// TIA Portal V16 export
// export: Created 2021-04-06T19:52:15.2153199Z, ExportSetting WithDefaults, DisplayName Totally Integrated Automation Portal, DisplayVersion V16, DisplayName TIA Portal Version Control Interface, DisplayVersion V16, DisplayName TIA Portal Openness, DisplayVersion V16, DisplayName STEP 7 Professional, DisplayVersion V16, DisplayName STEP 7 Safety, DisplayVersion V16, DisplayName WinCC Unified SCADA Engineering System, DisplayVersion V16
FUNCTION_BLOCK "modbus_SenecaConnectPort1"   // FB11, LAD
{ S7_Optimized_Access := 'TRUE' }
VERSION : 0.1
// stored: AutoNumber true, IsIECCheckEnabled false, IsRetainMemResEnabled false, MemoryReserve 100, SetENOAutomatically false, UDAEnableTagReadback false
   VAR_INPUT
      port : PORT;   // порт для подключения
      arrayAddressModbus : Array[0..12] of UInt;
      Offset_array_bits : SInt;
   END_VAR
   VAR_IN_OUT
      calibrateZero : Array[0..12] of Bool;
      taraZero : Array[0..12] of Bool;
      currentWeight : Array[0..12] of Real;
   END_VAR
   VAR
      MB_COMM_LOAD { S7_SetPoint := 'True'} : MB_COMM_LOAD;
      MB_MASTER { S7_SetPoint := 'True'} : MB_MASTER;
      Seneca : Struct
         TON_changeStep : TON_TIME;
         TON_Start { S7_SetPoint := 'True'} : Bool;
         "Step" : SInt;
      END_STRUCT;
      tmpWeight : Array[0..12] of DWord;
      restartPort : Bool;   // перезагрузка Modbus
   END_VAR
   VAR_TEMP
      index : SInt;
      tmpIndex : SInt;
   END_VAR
BEGIN

REGION Network 1: ИНИЦИАЛИЗИРУЕМ ПОРТ
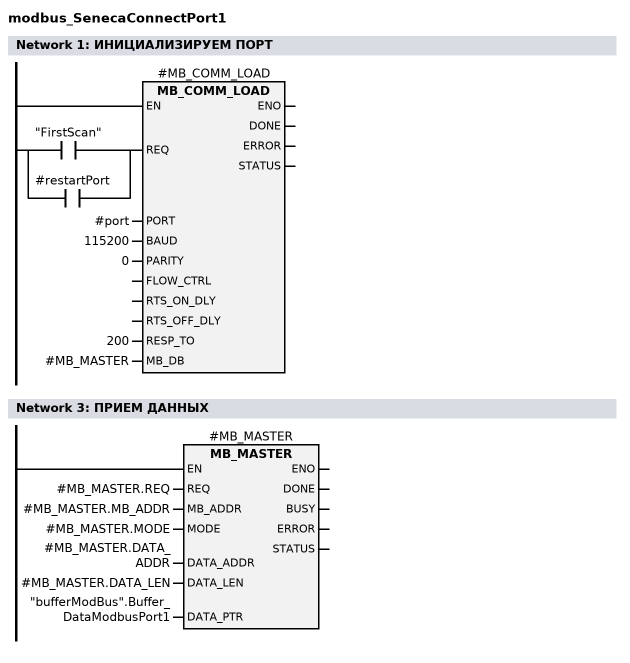
   RUNG wire#powerrail
      #MB_COMM_LOAD.MB_COMM_LOAD(REQ := wire#w1, PORT := #port, BAUD := 115200, PARITY := 0, FLOW_CTRL :=, RTS_ON_DLY :=, RTS_OFF_DLY :=, RESP_TO := 200, MB_DB := #MB_MASTER, DONE =>, ERROR =>, STATUS =>)
   END_RUNG
   RUNG wire#powerrail
      Contact( "FirstScan" )
   END_RUNG wire#w1
   RUNG wire#powerrail
      Contact( #restartPort )
   END_RUNG wire#w1
   // the same network as SCL:
   #MB_COMM_LOAD(REQ := "FirstScan" OR #restartPort,   // MB_COMM_LOAD
                 PORT := #port,
                 BAUD := 115200,
                 PARITY := 0,
                 RESP_TO := 200,
                 MB_DB := #MB_MASTER);
END_REGION

REGION Network 2 (SCL): ОБМЕН
   #Seneca.TON_changeStep(IN :=#Seneca.TON_Start,
                          PT := t#15ms);

   CASE #Seneca.Step OF

       1:
           #Seneca.Step := #Seneca.Step + 1;

       2: //ЧИТАЕМ ЗНАЧЕНИЕ ВЕСА С ПЕРВОГО МОДУЛЯ

           #index := 1+#Offset_array_bits;//заполнять функцию будем через индекс чтобы меньше писать
           "rcvDataWeight"(ADDR_DEVICE := #arrayAddressModbus[#index],
                           Ton_changeStep:=#Seneca.TON_changeStep,
                           Ton_Start:=#Seneca.TON_Start,
                           "Step":=#Seneca.Step,
                           MB_MASTER:=#MB_MASTER);

       3://ЧИТАЕМ ЗНАЧЕНИЕ ВЕСА СО ВТОРОГО МОДУЛЯ
           #index := 2+#Offset_array_bits;//заполнять функцию будем через индекс чтобы меньше писать
           "rcvDataWeight"(ADDR_DEVICE := #arrayAddressModbus[#index],
                           Ton_changeStep:=#Seneca.TON_changeStep,
                           Ton_Start:=#Seneca.TON_Start,
                           "Step":=#Seneca.Step,
                           MB_MASTER:=#MB_MASTER);

       4: // КАЛИБРОВКА 0 ДЛЯ ПЕРВОГО МОДУЛЯ и ТАРИРОВАНИЕ
           #index := 1+#Offset_array_bits;//заполнять функцию будем через индекс чтобы меньше писать
           "sndCALIBR&Tara"(ADDR_DEVICE := #arrayAddressModbus[#index],
                        ton_changeStep:=#Seneca.TON_changeStep,
                        MB_MASTER:=#MB_MASTER,
                        Ton_Start:=#Seneca.TON_Start,
                        Calibrate:=#calibrateZero[#index],
                        Buffer:="bufferModBus".Buffer_DataModbusPort1,
                        "Step":=#Seneca.Step,
                        Tara:=#taraZero[#index]);

       5:// КАЛИБРОВКА 0 ДЛЯ ВТОРОГО МОДУЛЯ и ТАРИРОВАНИЕ
           #index := 2+#Offset_array_bits;//заполнять функцию будем через индекс чтобы меньше писать
           "sndCALIBR&Tara"(ADDR_DEVICE := #arrayAddressModbus[#index],
                        ton_changeStep := #Seneca.TON_changeStep,
                        MB_MASTER := #MB_MASTER,
                        Ton_Start := #Seneca.TON_Start,
                        Calibrate := #calibrateZero[#index],
                        Buffer := "bufferModBus".Buffer_DataModbusPort1,
                        "Step" := #Seneca.Step,
                        Tara := #taraZero[#index]);

           //////////////////////////////////////////////////////////////////////////////////
           //////////////////////////////////////////////////////////////////////////////////
           //////////////////////////////////////////////////////////////////////////////////
           //////////////////////////////////////////////////////////////////////////////////
       6: //ЧИТАЕМ ЗНАЧЕНИЕ ВЕСА С ТРЕТЬЕГО МОДУЛЯ

           #index := 3+#Offset_array_bits;//заполнять функцию будем через индекс чтобы меньше писать
           "rcvDataWeight"(ADDR_DEVICE := #arrayAddressModbus[#index],
                           Ton_changeStep := #Seneca.TON_changeStep,
                           Ton_Start := #Seneca.TON_Start,
                           "Step" := #Seneca.Step,
                           MB_MASTER := #MB_MASTER);

       7://ЧИТАЕМ ЗНАЧЕНИЕ ВЕСА С ЧЕТВЕРТОГО МОДУЛЯ
           #index := 4+#Offset_array_bits;//заполнять функцию будем через индекс чтобы меньше писать
           "rcvDataWeight"(ADDR_DEVICE := #arrayAddressModbus[#index],
                           Ton_changeStep := #Seneca.TON_changeStep,
                           Ton_Start := #Seneca.TON_Start,
                           "Step" := #Seneca.Step,
                           MB_MASTER := #MB_MASTER);

       8:// КАЛИБРОВКА 0 ДЛЯ ТРЕТЬЕГО  МОДУЛЯ

           #index := 3+#Offset_array_bits;//заполнять функцию будем через индекс чтобы меньше писать
           "sndCALIBR&Tara"(ADDR_DEVICE := #arrayAddressModbus[#index],
                        ton_changeStep := #Seneca.TON_changeStep,
                        MB_MASTER := #MB_MASTER,
                        Ton_Start := #Seneca.TON_Start,
                        Calibrate := #calibrateZero[#index],
                        Buffer := "bufferModBus".Buffer_DataModbusPort1,
                        "Step" := #Seneca.Step,
                        Tara := #taraZero[#index]);

       9://КАЛИБРОВКА 0 ДЛЯ ЧЕТВЕРТОГО МОДУЛЯ

           #index := 4+#Offset_array_bits;//заполнять функцию будем через индекс чтобы меньше писать
           "sndCALIBR&Tara"(ADDR_DEVICE := #arrayAddressModbus[#index],
                        ton_changeStep := #Seneca.TON_changeStep,
                        MB_MASTER := #MB_MASTER,
                        Ton_Start := #Seneca.TON_Start,
                        Calibrate := #calibrateZero[#index],
                        Buffer := "bufferModBus".Buffer_DataModbusPort1,
                        "Step" := #Seneca.Step,
                        Tara := #taraZero[#index]);

           /////////////////////////////////////////////////////////////////////////////////
           ////////////////////////////////////////////////////////////////////////////////
           ////////////////////////////////////////////////////////////////////////////////
           ////////////////////////////////////////////////////////////////////////////////
       10: //ЧИТАЕМ ЗНАЧЕНИЕ ВЕСА С ПЯТОГО МОДУЛЯ
           #index := 5+#Offset_array_bits;//заполнять функцию будем через индекс чтобы меньше писать
           "rcvDataWeight"(ADDR_DEVICE := #arrayAddressModbus[#index],
                           Ton_changeStep := #Seneca.TON_changeStep,
                           Ton_Start := #Seneca.TON_Start,
                           "Step" := #Seneca.Step,
                           MB_MASTER := #MB_MASTER);

       11://ЧИТАЕМ ЗНАЧЕНИЕ ВЕСА С ШЕСТОГО МОДУЛЯ
           #index := 6+#Offset_array_bits;//заполнять функцию будем через индекс чтобы меньше писать
           "rcvDataWeight"(ADDR_DEVICE := #arrayAddressModbus[#index],
                           Ton_changeStep := #Seneca.TON_changeStep,
                           Ton_Start := #Seneca.TON_Start,
                           "Step" := #Seneca.Step,
                           MB_MASTER := #MB_MASTER);

       12:// КАЛИБРОВКА 0 ДЛЯ ПЯТОГО  МОДУЛЯ

           #index := 5+#Offset_array_bits;//заполнять функцию будем через индекс чтобы меньше писать
           "sndCALIBR&Tara"(ADDR_DEVICE := #arrayAddressModbus[#index],
                        ton_changeStep := #Seneca.TON_changeStep,
                        MB_MASTER := #MB_MASTER,
                        Ton_Start := #Seneca.TON_Start,
                        Calibrate := #calibrateZero[#index],
                        Buffer := "bufferModBus".Buffer_DataModbusPort1,
                        "Step" := #Seneca.Step,
                        Tara := #taraZero[#index]);

       13:// КАЛИБРОВКА 0 ДЛЯ ШЕСТОГО МОДУЛЯ
           #index := 6+#Offset_array_bits;//заполнять функцию будем через индекс чтобы меньше писать
           "sndCALIBR&Tara"(ADDR_DEVICE := #arrayAddressModbus[#index],
                        ton_changeStep := #Seneca.TON_changeStep,
                        MB_MASTER := #MB_MASTER,
                        Ton_Start := #Seneca.TON_Start,
                        Calibrate := #calibrateZero[#index],
                        Buffer := "bufferModBus".Buffer_DataModbusPort1,
                        "Step" := #Seneca.Step,
                        Tara := #taraZero[#index]);
   14://отправка аналоговых значений вибрации
       "sndVibration"(ADDR_DEVICE:=40,
                      ton_changeStep:= #Seneca.TON_changeStep,
                      MB_MASTER:=#MB_MASTER,
                      Ton_Start:=#Seneca.TON_Start,
                      Buffer:="bufferModBus".Buffer_DataModbusPort1,
                      "Step":=#Seneca.Step);

       ELSE
           #Seneca.Step := 1;
   END_CASE;
END_REGION

REGION Network 3: ПРИЕМ ДАННЫХ
   RUNG wire#powerrail
      #MB_MASTER.MB_MASTER(REQ := #MB_MASTER.REQ, MB_ADDR := #MB_MASTER.MB_ADDR, MODE := #MB_MASTER.MODE, DATA_ADDR := #MB_MASTER.DATA_ADDR, DATA_LEN := #MB_MASTER.DATA_LEN, DATA_PTR := "bufferModBus".Buffer_DataModbusPort1, DONE =>, BUSY =>, ERROR =>, STATUS =>)
   END_RUNG
   // the same network as SCL:
   #MB_MASTER(REQ := #MB_MASTER.REQ,   // MB_MASTER
              MB_ADDR := #MB_MASTER.MB_ADDR,
              MODE := #MB_MASTER.MODE,
              DATA_ADDR := #MB_MASTER.DATA_ADDR,
              DATA_LEN := #MB_MASTER.DATA_LEN,
              DATA_PTR := "bufferModBus".Buffer_DataModbusPort1);
END_REGION

REGION Network 4 (SCL)
   IF #Seneca.Step = 2 AND #MB_MASTER.DONE THEN
       #tmpIndex := 1 + #Offset_array_bits;
       #tmpWeight[#tmpIndex].%W0 := "bufferModBus".Buffer_DataModbusPort1[1];
       #tmpWeight[#tmpIndex].%W1 := "bufferModBus".Buffer_DataModbusPort1[0];
       #currentWeight[#tmpIndex] := DWORD_TO_REAL(#tmpWeight[#tmpIndex]);
       "bufferModBus".Buffer_DataModbusPort1[0] := 0;
       "bufferModBus".Buffer_DataModbusPort1[1] := 0;

   END_IF;

   IF #Seneca.Step = 3 AND #MB_MASTER.DONE THEN
       #tmpIndex := 2 + #Offset_array_bits;
       #tmpWeight[#tmpIndex].%W0 := "bufferModBus".Buffer_DataModbusPort1[1];
       #tmpWeight[#tmpIndex].%W1 := "bufferModBus".Buffer_DataModbusPort1[0];
       #currentWeight[#tmpIndex] := DWORD_TO_REAL(#tmpWeight[#tmpIndex]);
       "bufferModBus".Buffer_DataModbusPort1[0] := 0;
       "bufferModBus".Buffer_DataModbusPort1[1] := 0;
   END_IF;

   IF #Seneca.Step = 6 AND #MB_MASTER.DONE THEN
       #tmpIndex := 3 + #Offset_array_bits;
       #tmpWeight[#tmpIndex].%W0 := "bufferModBus".Buffer_DataModbusPort1[1];
       #tmpWeight[#tmpIndex].%W1 := "bufferModBus".Buffer_DataModbusPort1[0];
       #currentWeight[#tmpIndex] := DWORD_TO_REAL(#tmpWeight[#tmpIndex]);
       "bufferModBus".Buffer_DataModbusPort1[0] := 0;
       "bufferModBus".Buffer_DataModbusPort1[1] := 0;
   END_IF;

   IF #Seneca.Step = 7 AND #MB_MASTER.DONE THEN
       #tmpIndex := 4 + #Offset_array_bits;
       #tmpWeight[#tmpIndex].%W0 := "bufferModBus".Buffer_DataModbusPort1[1];
       #tmpWeight[#tmpIndex].%W1 := "bufferModBus".Buffer_DataModbusPort1[0];
       #currentWeight[#tmpIndex] := DWORD_TO_REAL(#tmpWeight[#tmpIndex]);
       "bufferModBus".Buffer_DataModbusPort1[0] := 0;
       "bufferModBus".Buffer_DataModbusPort1[1] := 0;
   END_IF;

   IF #Seneca.Step = 10 AND #MB_MASTER.DONE THEN
       #tmpIndex := 5 + #Offset_array_bits;
       #tmpWeight[#tmpIndex].%W0 := "bufferModBus".Buffer_DataModbusPort1[1];
       #tmpWeight[#tmpIndex].%W1 := "bufferModBus".Buffer_DataModbusPort1[0];
       #currentWeight[#tmpIndex] := DWORD_TO_REAL(#tmpWeight[#tmpIndex]);
       "bufferModBus".Buffer_DataModbusPort1[0] := 0;
       "bufferModBus".Buffer_DataModbusPort1[1] := 0;
   END_IF;

   IF #Seneca.Step = 11 AND #MB_MASTER.DONE THEN
       #tmpIndex := 6 + #Offset_array_bits;
       #tmpWeight[#tmpIndex].%W0 := "bufferModBus".Buffer_DataModbusPort1[1];
       #tmpWeight[#tmpIndex].%W1 := "bufferModBus".Buffer_DataModbusPort1[0];
       #currentWeight[#tmpIndex] := DWORD_TO_REAL(#tmpWeight[#tmpIndex]);
       "bufferModBus".Buffer_DataModbusPort1[0] := 0;
       "bufferModBus".Buffer_DataModbusPort1[1] := 0;
   END_IF;
END_REGION
END_FUNCTION_BLOCK
